Universal Robots PolyScope program: joyControl.urp

Program joyControl (installation=default directory=/programs/bcastets createdIn=3.10.0.76181 lastSavedIn=3.10.0.76181 robotSerialNumber=2016352450)
Calibrated DH parameters: a=[0.000246, -0.041637, -0.381793, 0.000071, 0.000086, 0]; d=[0.089255, 475.628349, -451.442723, -24.075242, 0.094834, 0.082514]; alpha=[1.5703, -0.000889, -0.003696, 1.569893, -1.570803, 0]; deltaTheta=[0.000008, -1.472641, 1.242698, 0.230075, -0.000006, 0.000032]
BeforeStart
  MoveJ speed 60 deg/s, acceleration 80 deg/s^2 (useActiveTCP=true)
    Waypoint home: TCP in base x=349.217 y=-141.392 z=524.16 mm, rx=-1.3478 ry=1.1309 rz=-1.2935 rad; joints [-6.733, -75.487, -114.677, 8.817, 98.032, -9.216] deg
Robot Program (runOnlyOnce=false)
  startPose := get_actual_tcp_pose()
  r := d2r(5*(L_upDown-100)/100)
  p := d2r(5*(L_leftRright-100)/100)
  yaw := d2r(5*(R_leftRight-100)/100)
  rVector := rpy2rotvec([r,p,yaw])
  rx := rVector[0]
  ry := rVector[1]
  rz := rVector[2]
  startPose := pose_trans(startPose,p[0,0,0,rx,ry,rz])
  endPose := pose_trans(startPose,p[0,0,-0.05*(R_upDown-100)/100,0,0,0])
  MoveJ speed 60 deg/s, acceleration 80 deg/s^2 (useActiveTCP=true)
    Waypoint Waypoint_1 (Variable): variable=endPose
  Script: stopj(20)
  Wait Sleep waitTime=0.1
